// TIA Portal V18 export
FUNCTION "AIbasic" : Void   // FC10001, FBD
{ S7_Optimized_Access := 'TRUE' }
VERSION : 0.1
// stored: AutoNumber false, IsIECCheckEnabled false, SetENOAutomatically false, UDAEnableTagReadback false
   VAR_INPUT
      iInput : Int;
      iFilterValue : Int;
      rMin : Real;
      rMax : Real;
   END_VAR
   VAR_OUTPUT
      rOutput : Real;
      iOutput : Int;
   END_VAR
   VAR_TEMP
      rNorm : Real;
      rOut : Real;
      rOut_real : Real;
   END_VAR
BEGIN

REGION Network 1
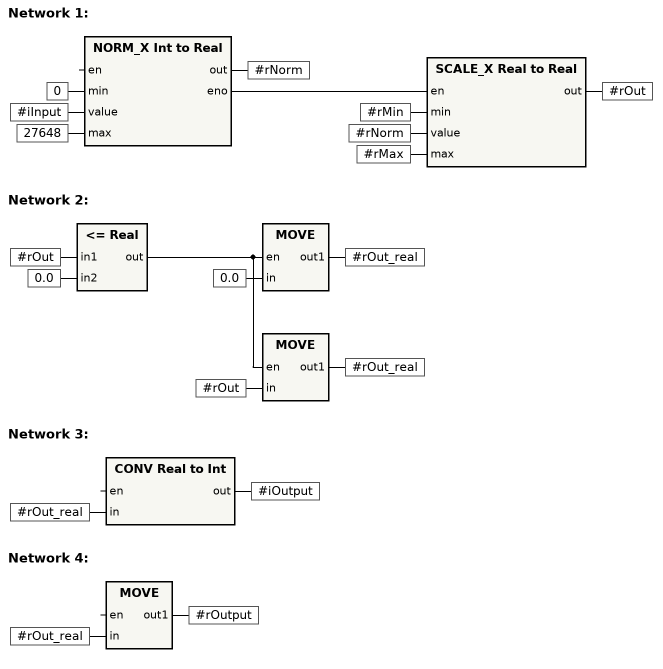
   #rNorm := NORM_X(MIN := 0, VALUE := #iInput, MAX := 27648);
   #rOut := SCALE_X(MIN := #rMin, VALUE := #rNorm, MAX := #rMax);
END_REGION

REGION Network 2
   IF #rOut <= 0.0 THEN
       #rOut_real := 0.0;
       #rOut_real := #rOut;
   END_IF;
END_REGION

REGION Network 3
   #iOutput := REAL_TO_INT(#rOut_real);
END_REGION

REGION Network 4
   #rOutput := #rOut_real;
END_REGION
END_FUNCTION
